{attribute 'linkalways'} 
{attribute 'no_explicit_call' := 'This FB is a CLASS and must be accessed using methods or properties'}
{attribute 'enable_dynamic_creation'}
FUNCTION_BLOCK _ETcVnBoostClassifierType EXTENDS EnumDatatypeBase
VAR
	localData : ETcVnBoostClassifierType;
	activeData : REFERENCE TO ETcVnBoostClassifierType;
	enumBaseDatatype : _DINT(localData);
END_VAR

METHOD PRIVATE AddLocalEnumeration
VAR_INPUT
	Enumeration : T_MAXSTRING;
	Value : ETcVnBoostClassifierType;
END_VAR
AddEnumeration(Enumeration, Value);
END_METHOD

PROPERTY PUBLIC Address : PVOID
GET
Address := ADR(activeData);
END_GET
END_PROPERTY

METHOD PUBLIC ClearReference
VAR_INPUT
END_VAR
activeData REF= localData;
SetBaseDatatypeReference();
END_METHOD

METHOD PUBLIC Clone : I_Datatype
VAR
    pClone : POINTER TO _ETcVnBoostClassifierType;
END_VAR
pClone := __NEW(_ETcVnBoostClassifierType(InitialValue := Value));
Clone := pClone^;
END_METHOD

METHOD FB_init : BOOL
VAR_INPUT
	bInitRetains : BOOL; // if TRUE, the retain variables are initialized (warm start / cold start)
	bInCopyCode : BOOL;  // if TRUE, the instance afterwards gets moved into the copy code (online change)
	InitialValue : ETcVnBoostClassifierType;
END_VAR
localData := InitialValue;
AddBaseDatatype(enumBaseDatatype);
ClearReference();

AddLocalEnumeration('TCVN_BCT_DISCRETE', ETcVnBoostClassifierType.TCVN_BCT_DISCRETE);
AddLocalEnumeration('TCVN_BCT_REAL', ETcVnBoostClassifierType.TCVN_BCT_REAL);
AddLocalEnumeration('TCVN_BCT_LOGIT', ETcVnBoostClassifierType.TCVN_BCT_LOGIT);
AddLocalEnumeration('TCVN_BCT_GENTLE', ETcVnBoostClassifierType.TCVN_BCT_GENTLE);
END_METHOD

PROPERTY PUBLIC Identifier : T_MAXSTRING
GET
Identifier := 'ETcVnBoostClassifierType';
END_GET
END_PROPERTY

METHOD IsEnumeratorValueEqual : BOOL
VAR_INPUT
	Enumerator : I_KeyValueForwardEnumerator;
END_VAR
VAR
	storedValue : ETcVnBoostClassifierType;
END_VAR
IF NOT Enumerator.TryGet(storedValue) THEN
	RETURN;
END_IF

IsEnumeratorValueEqual := storedValue = activeData;
END_METHOD

METHOD PUBLIC MakeReferenceTo
VAR_INPUT
	ReferenceTarget : REFERENCE TO ETcVnBoostClassifierType;
END_VAR
activeData REF= ReferenceTarget;
SetBaseDatatypeReference();
END_METHOD

METHOD PROTECTED SetBaseDatatypeReference
VAR_INPUT
END_VAR
enumBaseDatatype.MakeReferenceTo(activeData);
END_METHOD

PROPERTY PUBLIC Size : UDINT
GET
Size := SIZEOF(activeData);
END_GET
END_PROPERTY

METHOD TryMakeReferenceTo : BOOL
VAR_INPUT
	Target : I_Datatype;
END_VAR
VAR
	pTargetData : POINTER TO ETcVnBoostClassifierType;
END_VAR
IF NOT IsEquivalentTo(Target) THEN
	RETURN;
END_IF

pTargetData := Target.Address;
activeData REF= pTargetData^;
SetBaseDatatypeReference();
TryMakeReferenceTo := TRUE;
END_METHOD

PROPERTY PUBLIC Value : ETcVnBoostClassifierType
GET
Value := activeData;
END_GET
SET
activeData := Value;
END_SET
END_PROPERTY

END_FUNCTION_BLOCK

(* stored: Version 1.1.0.1, ProductVersion 3.1.4024.13
   POU _ETcVnBoostClassifierType: Id {d7b79db4-ab1c-009e-172b-0883b9fbbe0d}, SpecialFunc None
   Folder Core: Id {240e84cc-f842-07b0-1f9f-6bd659207f5f}
   Folder Protected: Id {4dd4ede2-4bb2-00f9-2886-25e9b66ed7cc}
   Folder Customize: Id {81c0cb85-0763-0e4e-311d-47f0eafa052d}
   Folder Constructor: Id {d3affc3e-1f32-0107-107e-98f20e45a264}
   Folder Private: Id {362183d3-c265-0640-1dd6-68809b2980f8}
   Folder Protected: Id {3e9c7f48-0fe6-0ab2-1d6f-32d297926bf3}
   Method AddLocalEnumeration: Id {7654df0f-771a-005f-0aa8-5777765faeb0}
   Property Address: Id {033617ab-0d16-0c09-2a8c-411290034410}
   Get Get: Id {87fcb994-373b-0845-39b6-649607bb0151}
   Method ClearReference: Id {eb6e2b6b-fd0a-016c-372f-36288195f561}
   Method Clone: Id {36f2d384-b25b-0865-373b-1f48ca1dae27}
   Method FB_init: Id {b1cd6443-3f62-0495-15e6-728c7e47e0b2}
   Property Identifier: Id {fe48173f-2ab7-0a40-3643-f1bd3be8f31d}
   Get Get: Id {820c2bd4-eace-031b-28ab-2921f0451684}
   Method IsEnumeratorValueEqual: Id {6380ab07-dc4c-039e-2340-11ba7b3a05ae}
   Method MakeReferenceTo: Id {e25c9ede-44fd-00cf-3ae2-bdb9e78782cf}
   Method SetBaseDatatypeReference: Id {aed47cf4-4846-0389-3c33-21dbf982b38d}
   Property Size: Id {dd5fbab4-da81-0f80-2b0b-219904f6675e}
   Get Get: Id {583b0d43-3317-03a3-13ac-d4fd47e8a8a1}
   Method TryMakeReferenceTo: Id {ac81e19d-7693-066e-031d-3da2ddcb028b}
   Property Value: Id {ebf58b05-92ca-0856-2f52-d2790805b5db}
   Get Get: Id {1a118f57-5887-0383-0c0d-6ab9fb7605ba}
   Set Set: Id {dbdefce1-e138-00dc-1ad6-fd7492bb060c} *)
